# EPICS substitutions: template/others_type1_ess.substitutions
global {dev=$(dev)}

file "fru_common_ess.template"
{
   pattern { id		, unit	, fruid	}
           { SH		, 1  	, 1	}
           { SH		, 2  	, 2	}
           { CM		, 1  	, 253	}
           { SHM	, 1  	, 254	}
}
